// TIA Portal project "Baume" (V12)

(* hardware
DEVICE "S7-1200 station_2"  SIMATIC 1200-Station
   slot 0: "S7-1200 rack"  Rack  V1.0
   slot 1: "PLC_1"  CPU 1212C DC/DC/Rly  6ES7 212-1HD30-0XB0  V1.0
   slot 101: "CM 1241 (RS422/485)_1"  6ES7 241-1CH32-0XB0  V2.0
*)

// ===== PLC "PLC_1"  CPU 1212C DC/DC/Rly =====

VAR_GLOBAL   // PLC tag table "Default tag table"
   "Empty_level" AT %M0.1 : Bool;
   "Tag_9(1)" AT %MW10 : Word;
   "Tag_1" AT %MW30 : Word;
   "Tag_2" AT %MD12 : Time;
   "Tag_3" AT %MD20 : Time;
   "Tag_4" AT %IW256 : Word;
   "Tag_5" AT %M5.0 : Bool;
   "percentage" AT %MW20 : Word;
   "percentage_real" AT %MD4 : Real;
   "Tag_7" AT %M6.0 : Bool;
   "Tag_6" AT %MD17 : Real;
   "Tag_8" AT %MW15 : Int;
   "Output_0-20mA" AT %MW5 : Int;
   "Output_4-20mA" AT %MW8 : Int;
   "Tag_9" AT %Q0.0 : Bool;
   "Caustic_valve" AT %Q0.1 : Bool;
   "Medium_level" AT %M0.2 : Bool;
   "Water_valve" AT %Q0.2 : Bool;
   "timer_1" AT %MD10 : Time;
   "High_level" AT %M0.3 : Bool;
   "timer_2" AT %MD14 : Time;
   "Start" AT %M0.0 : Bool;
   "Tag_10" AT %MD5 : Real;
END_VAR

// folder: System blocks/Program resources

DATA_BLOCK "timer_01"   // DB1
{ S7_Optimized_Access := 'FALSE' }
AUTHOR : Simatic
FAMILY : IEC
NAME : IEC_TMR
VERSION : 1.0
// stored: InstanceOfName ?
"?"
BEGIN
END_DATA_BLOCK

DATA_BLOCK "timer_02"   // DB2
{ S7_Optimized_Access := 'FALSE' }
AUTHOR : Simatic
FAMILY : IEC
NAME : IEC_TMR
VERSION : 1.0
// stored: InstanceOfName ?
"?"
BEGIN
END_DATA_BLOCK

// folder: (top level)

FUNCTION "0-20 to 4-20mA" : Void   // FC1, LAD
{ S7_Optimized_Access := 'FALSE' }
VERSION : 0.1
   VAR_INPUT
      "Input_0-20mA" : Int;
   END_VAR
   VAR_OUTPUT
      "Output_4-20mA" : Int;
   END_VAR
   VAR_TEMP
      Temp_input_real : Real;
      Temp_analog_real : Real;
   END_VAR
BEGIN

REGION Network 1
   // 27648-5529.6=(22118.4)*x1=x*22118.4   where 5529.6-<Zero (4-20mA)
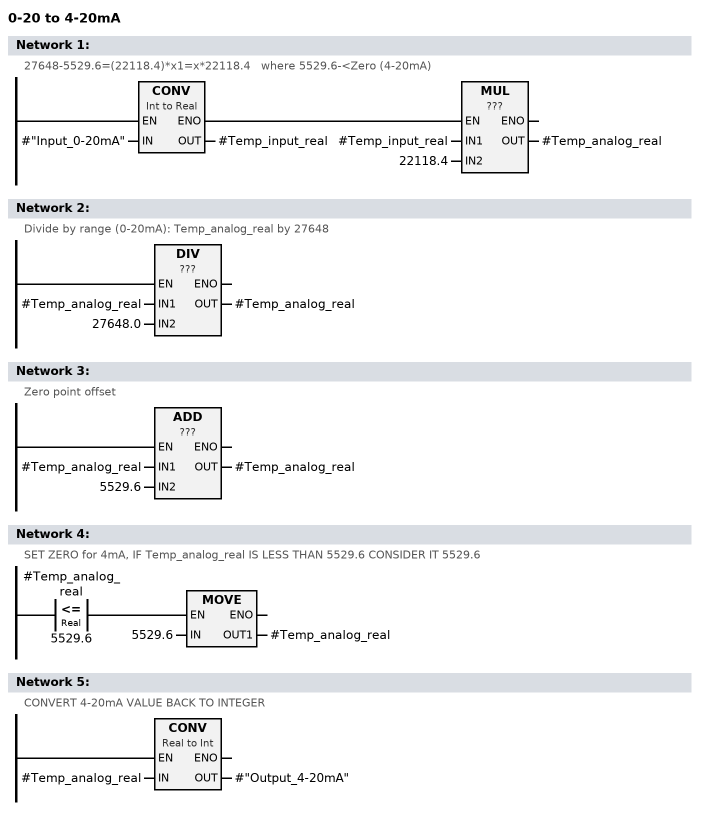
   RUNG wire#powerrail
      { S7_Templates := "[SrcType := Int, DestType := Real]"; S7_GenerateENO := "TRUE" } Convert(in := #"Input_0-20mA", out => #Temp_input_real)
      { S7_Templates := "SrcType := ???"; S7_GenerateENO := "TRUE" } Mul(in1 := #Temp_input_real, in2 := 22118.4, out => #Temp_analog_real)
   END_RUNG
   // the same network as SCL:
   // ENO of a box is taken as its EN; it also drops when the box reports an error
   #Temp_input_real := INT_TO_REAL(#"Input_0-20mA");
   #Temp_analog_real := #Temp_input_real * 22118.4;
END_REGION

REGION Network 2
   // Divide by range (0-20mA): Temp_analog_real by 27648
   RUNG wire#powerrail
      { S7_Templates := "SrcType := ???"; S7_GenerateENO := "TRUE" } Div(in1 := #Temp_analog_real, in2 := 27648.0, out => #Temp_analog_real)
   END_RUNG
   // the same network as SCL:
   #Temp_analog_real := #Temp_analog_real / 27648.0;
END_REGION

REGION Network 3
   // Zero point offset
   RUNG wire#powerrail
      { S7_Templates := "SrcType := ???"; S7_GenerateENO := "TRUE" } Add(in1 := #Temp_analog_real, in2 := 5529.6, out => #Temp_analog_real)
   END_RUNG
   // the same network as SCL:
   #Temp_analog_real := #Temp_analog_real + 5529.6;
END_REGION

REGION Network 4
   // SET ZERO for 4mA, IF Temp_analog_real IS LESS THAN 5529.6 CONSIDER IT 5529.6
   RUNG wire#powerrail
      { S7_Templates := "SrcType := Real" } LE_Contact(in1 := #Temp_analog_real, in2 := 5529.6)
      { S7_GenerateENO := "TRUE" } Move(in := 5529.6, out1 => #Temp_analog_real)
   END_RUNG
   // the same network as SCL:
   IF #Temp_analog_real <= 5529.6 THEN #Temp_analog_real := 5529.6; END_IF;
END_REGION

REGION Network 5
   // CONVERT 4-20mA VALUE BACK TO INTEGER
   RUNG wire#powerrail
      { S7_Templates := "[SrcType := Real, DestType := Int]"; S7_GenerateENO := "TRUE" } Convert(in := #Temp_analog_real, out => #"Output_4-20mA")
   END_RUNG
   // the same network as SCL:
   #"Output_4-20mA" := REAL_TO_INT(#Temp_analog_real);
END_REGION
END_FUNCTION

ORGANIZATION_BLOCK "Main"   // OB1, LAD, ProgramCycle
TITLE = "Main Program Sweep (Cycle)"
{ S7_Optimized_Access := 'FALSE' }
VERSION : 0.1
BEGIN
END_ORGANIZATION_BLOCK